TYPE ST_AteqValveMap :
STRUCT
    nValveStartIndex : UINT;    // starting bit position in the full valve bank
    nNumOfValves     : UINT;    // number of valves this ATEQ uses
END_STRUCT
END_TYPE

(* stored: Version 1.1.0.1
   DUT ST_AteqValveMap: Id {71c12f32-aa8f-43e0-bf1d-88be6427ca2f} *)
